(* CODESYS project festo_vtem_devcon_v3.5.7.235.library
   Version: 3.5.7.235
   Author: JEBU/MKLP
   Description: Festo VTEM device controlling functions interface
   Title: Festo_VTEM_DevCon
   DefaultNamespace: FestoVTEMdc
   LanguageModelAttribute: qualified-access-only
   Company: Festo SE & Co. KG

Project tree, tasks and I/O mapping:
  data type eValveState
  auxiliary Functions/
    function block FB_Read_Bits_From_Word [ST]
    function block FB_Write_Value_To_Word [ST]
    function block FB_Read_Bits_From_Byte [ST]
  StateInterpreter/
    function block FB_StateInterpreter_MA_07 [ST]
    function block FB_StateInterpreter_MA_01 [ST]
    function block FB_StateInterpreter_MA_11 [ST]
    function block FB_StateInterpreter_MA_12 [ST]
    function block FB_StateInterpreter_MA_06 [ST]
    function block FB_StateInterpreter_MA_02 [ST]
    function block FB_StateInterpreter_MA_03 [ST]
    function block FB_StateInterpreter_MA_04 [ST]
    function block FB_StateInterpreter_MA_05 [ST]
    function block FB_StateInterpreter_MA_08 [ST]
    function block FB_StateInterpreter_MA_33 [ST]
    function block FB_StateInterpreter_TeachInRun [ST]
  Operation/
    data type eResponseToValveModeSet
    function block FB_ValveControl [ST]
    function block FB_TeachInRun [ST]
  Transfermode/
    data type eTransferResponse
    data type stTransferPackage
    specific_MA_config/
      function block FB_Write_config_MA_07 [ST]
      function block FB_Write_config_MA_04 [ST]
      function block FB_Write_config_MA_11 [ST]
      function block FB_Write_config_MA_12 [ST]
      function block FB_Write_config_MA_02 [ST]
      function block FB_Write_config_MA_03 [ST]
      function block FB_Write_config_MA_08 [ST]
      function block FB_Write_config_MA_05 [ST]
      function block FB_Write_config_MA_01 [ST]
      function block FB_Write_config_MA_06 [ST]
      function block FB_Write_config_MA_33 [ST]
    data type eSavingResponse
    data type stMalfunction
    function block FB_Download_Multiple_Parameters [ST]
    function block FB_Download_Single_Parameter [ST]
    function block FB_Upload_Multiple_Parameters [ST]
    function block FB_Upload_Single_Parameter [ST]
    function block FB_Save_Configuration_Persistent [ST]
    function block FB_Write_config_AI_Module [ST]
    function block FB_Write_config_DI_Module [ST]
    function block FB_ReadMalfunctionList [ST]
  data type eValveMode
  data type eResponseTeachInRun
  data type eResponseReadMalfunctionList
*)

// Operation/eResponseToValveModeSet
(*****************************************************************************************************

Festo SE & Co. KG, Esslingen
Copyright (c) 2019. All rights reserved.

Product:            Motion Terminal VTEM
Description:        Enum for responding values sent by the Motion Terminal or the function blocks

Object version:     1.01
Last change:        2019
======================================================================================================
                                       H I S T O R Y
======================================================================================================
Version:            1.01
Date:               2019-04
Change/Activity:    - added new Value "FB_not_enabled := 1051"
Release:            3.5.7.232
Author:             MKLP
------------------------------------------------------------------------------------------------------
Version:            1.00
Date:               2017
Change/Activity:    - created
Release:            3.5.7.220
Author:             HLBG
======================================================================================================

*****************************************************************************************************)

TYPE eResponseToValveModeSet :
(
	// info provided by Motion Terminal protocol ("app state")
	reserved 								:= 0,
	invalid_SetValveMode 					:= 1,
	invalid_SetAppControl 					:= 2,
	invalid_SetAppOption 					:= 3,
	invalid_SetPointValue1 					:= 4,
	invalid_SetPointValue2 					:= 5,
	invalid_configuration 					:= 6,

	access_denied_WebConfig 				:= 10,
	access_denied_saving_parameterisation 	:= 11,
	no_license_for_this_MA 					:= 12,
	all_licenses_in_use 					:= 13,
	invalid_license_file 					:= 14,
	no_valve_detected 						:= 15,
	valve_self_calibration_running 			:= 16,
	

	// additional FB internal info (not part of Motion Terminal protocol)
	no_TransferMode_with_this_FB			:= 1020,
	
	preparing_for_start 					:= 1031,
	starting 								:= 1032,
	MA_running 								:= 1033,
	TransferMode_running					:= 1034,
	stopping 								:= 1035,
	all_MAs_stopped 						:= 1036,
	acknowledge_needed 						:= 1037,
	failure 								:= 1038,

	preparing_for_acknowledge 				:= 1040,
	acknowledging 							:= 1041,
	all_errors_acknowledged 				:= 1042,
	failure_still_active 					:= 1043,

	no_communication 						:= 1050,
	FB_not_enabled							:= 1051
);
END_TYPE

// eValveState
(*****************************************************************************************************

Festo SE & Co. KG, Esslingen
Copyright (c) 2018. All rights reserved.

Product:            Motion Terminal VTEM
Description:        Enum to interpret the valve state value

Object version:     1.00
Last change:        2017
======================================================================================================
                                       H I S T O R Y
======================================================================================================
Version:            1.00
Date:               2017
Change/Activity:    - created
Release:            3.5.7.220
Author:             HLBG
======================================================================================================

*****************************************************************************************************)

TYPE eValveState :
(
	// info provided by Motion Terminal protocol ("valve state")
	NotReady 		:= 0, 
	Configurable 	:= 1, 
	Running 		:= 2,
	Failure 		:= 3
);
END_TYPE

// Transfermode/eTransferResponse
(*****************************************************************************************************

Festo SE & Co. KG, Esslingen
Copyright (c) 2018. All rights reserved.

Product:            Motion Terminal VTEM
Description:        Enum for responding values sent by the Motion Terminal or the function blocks

Object version:     1.03
Last change:        2020-03
======================================================================================================
                                       H I S T O R Y
======================================================================================================
Version:            1.03
Date:               2020-03
Change/Activity:    - added value 8 (#3104444)
Release:            not released yet
Author:             JEBU/MKLP
------------------------------------------------------------------------------------------------------
Version:            1.02
Date:               2018-11
Change/Activity:    - added values 29, 30 
Release:            3.5.7.233
Author:             JEBU
------------------------------------------------------------------------------------------------------
Version:            1.01
Date:               2018-08
Change/Activity:    - added values 27, 28 
Release:            3.5.7.221
Author:             JEBU
------------------------------------------------------------------------------------------------------
Version:            1.00
Date:               2017
Change/Activity:    - created
Release:            3.5.7.220
Author:             HLBG
======================================================================================================

*****************************************************************************************************)

TYPE eTransferResponse :
(
	// info provided by Motion Terminal protocol ("invalid command")
	reserved 								:= 0,
	invalid_Channel 						:= 1,
	invalid_TransferControl 				:= 2,
	invalid_AddressedTarget 				:= 3,
	invalid_Index 							:= 4,
	invalid_TransferValue 					:= 5,
	invalid_Combination 					:= 6,
	access_denied_DataInUse					:= 7,
	no_data_empty_slot						:= 8,
	
	// additional FB internal info (not part of Motion Terminal protocol)
	invalid_ParameterSet 					:= 9,
	
	// info provided by Motion Terminal protocol ("app state")
	access_denied_WebConfig 				:= 10,
	access_denied_saving 					:= 11,
	no_valve_detected 						:= 15,
	
	// additional FB internal info (not part of Motion Terminal protocol)
	reading_transfermode					:= 20,	
	ready_for_new_transfer 					:= 21,
	preparing_transfer 						:= 22,
	transferring 							:= 23,
	transfer_successful 					:= 24,
	FB_needs_rising_edge_xExecute			:= 25,
	Valve_Mode_is_not_61_inactive			:= 26,
	invalid_firmware_version				:= 27,
	communication_failed					:= 28,
	invalid_module_number					:= 29,
	resetting								:= 30
);
END_TYPE

// Transfermode/stTransferPackage
(*****************************************************************************************************

Festo SE & Co. KG, Esslingen
Copyright (c) 2018. All rights reserved.

Product:            Motion Terminal VTEM
Description:        Struct for transfer mode data

Object version:     1.00
Last change:        2017
======================================================================================================
                                       H I S T O R Y
======================================================================================================
Version:            1.00
Date:               2017
Change/Activity:    - created
Release:            3.5.7.220
Author:             HLBG
======================================================================================================

*****************************************************************************************************)

TYPE stTransferPackage :
	STRUCT
		iChannel			: INT;		(* the channel the value is to be written to (see documentation for details) *)
		iAddressedTarget	: INT; 		(* the target by which the parameter value is to be used (was "iAddressedApp" in former versions) (see documentation for details)*)
		iIndex				: INT; 		(* the index of the parameter (see documentation for details) *)
		iTransferValue		: INT; 		(* the value to be transfered *)
	END_STRUCT
END_TYPE

// Transfermode/eSavingResponse
(*****************************************************************************************************

Festo SE & Co. KG, Esslingen
Copyright (c) 2018. All rights reserved.

Product:            Motion Terminal VTEM
Description:        Enum for values sent back from the Motion Terminal during saving process 

Object version:     1.01
Last change:        2019-07
======================================================================================================
                                       H I S T O R Y
======================================================================================================
Version:            1.01
Date:               2019-07
Change/Activity:    - added value 25 "FB_needs_rising_edge_xExecute" (#2369163)
Release:            not released yet
Author:             JEBU/MKLP
------------------------------------------------------------------------------------------------------
Version:            1.00
Date:               2017
Change/Activity:    - created
Release:            3.5.7.220
Author:             HLBG
======================================================================================================

*****************************************************************************************************)

TYPE eSavingResponse :
(
	// info provided by Motion Terminal protocol (saving progress)
	reserved 				:= 0,
	saving_in_progress 		:= 1,
	saving_successful 		:= 2,
	saving_not_possible 	:= 3,
	saving_failed 			:= 4,
	
	// info provided by Motion Terminal protocol ("app state")
	access_denied_WebConfig := 10,
	access_denied_saving	:= 11,
	no_valve_detected 		:= 15,
	
	// additional FB internal info (not part of Motion Terminal protocol)
	preparing_to_save 		:= 20,
	ready_to_save 			:= 21,
	FB_needs_rising_edge_xExecute	:= 25
);
END_TYPE

// eValveMode
(*****************************************************************************************************

Festo SE & Co. KG, Esslingen
Copyright (c) 2018. All rights reserved.

Product:            Motion Terminal VTEM
Description:        Enum for values of the valve mode 

Object version:     1.01
Last change:        2020-04
======================================================================================================
                                       H I S T O R Y
======================================================================================================
Version:            1.01
Date:               2020-04
Change/Activity:    - created
Release:            3.5.7.234
Author:             JEBU
======================================================================================================

*****************************************************************************************************)

TYPE eValveMode :
(
	MA01_Directional_control_valve_functions							:= 1,
	MA02_Proportional_directional_control_valve							:= 2,
	MA03_Proportional_pressure_regulation								:= 3,
	MA04_Modelbased_proportional_pressure_regulation					:= 4,
	MA05_Supply_and_exhaust_air_flow_control							:= 5,
	MA06_ECO_drive														:= 6,
	MA07_Presetting_of_travel_time										:= 7,
	MA08_Selectable_pressure_level_ECO									:= 8,
	MA11_Soft_stop														:= 11,
	MA12_Leakage_diagnostics											:= 12,
	MA32_Positioning_and_Force											:= 32,
	MA33_Positioning													:= 33,
	VM60_TeachIn_run													:= 60,
	VM61_Inactive														:= 61,
	VM63_Transfermode													:= 63
);
END_TYPE

// Transfermode/stMalfunction
(*****************************************************************************************************

Festo SE & Co. KG, Esslingen
Copyright (c) 2018. All rights reserved.

Product:            Motion Terminal VTEM
Description:        Struct for complete entry in malfunction list (code, subcode, classification)

Object version:     1.00
Last change:        2018
======================================================================================================
                                       H I S T O R Y
======================================================================================================
Version:            1.00
Date:               2018
Change/Activity:    - created (#2256305)
Release:            not released yet
Author:             JEBU
======================================================================================================

*****************************************************************************************************)

TYPE stMalfunction :
STRUCT
	usiMalfunctionCode				: USINT;		// Malfunction Code
	usiMalfunctionSubcode			: USINT;		// Malfunction Subcode
	usiMalfunctionClassification	: USINT;		// Malfunction Classification
END_STRUCT
END_TYPE

// eResponseTeachInRun
(*****************************************************************************************************

Festo SE & Co. KG, Esslingen
Copyright (c) 2019. All rights reserved.
 
Product:            Motion Terminal VTEM
Description:        Enum status of the teach-in run process as it is displayed in the app state byte
 
Object version:     1.05
Last change:        2020-04
======================================================================================================
                                       H I S T O R Y
======================================================================================================
Version:            1.05
Date:               2020-04
Change/Activity:    - created (#2256363)
Release:            3.5.7.234
Author:             JEBU
======================================================================================================

******************************************************************************************************)

TYPE eResponseTeachInRun :
(
	// following entries correspond to the values of the AppState byte of the teach-in run
	TeachInRun_reserved								:= 0,
	TeachInRun_unlearned							:= 1,
	TeachInRun_check_tubes							:= 2,
	TeachInRun_choose_control						:= 3,
	TeachInRun_tune_trajectory						:= 4,
	TeachInRun_determine_reference_value			:= 5,
	TeachInRun_identification						:= 6,
	TeachInRun_partially_completed_only_2			:= 12,
	TeachInRun_partially_completed_only_4			:= 13,
	TeachInRun_completed							:= 14,
	TeachInRun_error								:= 15,
	
	// following entries are copies from eResponseToValveModeSet, their values are origins + 100	
	invalid_SetValveMode 							:= 101,
	invalid_SetAppControl 							:= 102,
	invalid_SetAppOption 							:= 103,
	invalid_SetPointValue1 							:= 104,
	invalid_SetPointValue2 							:= 105,
	invalid_configuration 							:= 106,
                                            	
	access_denied_WebConfig 						:= 110,
	access_denied_saving_parameterisation 			:= 111,
	no_license_for_this_MA 							:= 112,
	all_licenses_in_use 							:= 113,
	invalid_license_file 							:= 114,
	no_valve_detected 								:= 115,
	valve_self_calibration_running 					:= 116,
	
	// additional FB internal info (not part of Motion Terminal protocol)
	idle											:= 210,
	storing_first_cycle_input_data					:= 215,
	resetting_valve_to_61							:= 220,
	ReadingActiveParameterSet						:= 230,
	ChangingActiveParameterSet						:= 232,
	writing_parameter_MotionAppToBeToughtIn			:= 234,
	running_teachIn_run								:= 240,
	error_occured_check_DiagnosticMemory			:= 270,
	input_data_invalid								:= 271,
	FB_needs_rising_edge_xEnable					:= 272,
	acknowledge_needed								:= 273,
	Invalid_MotionAppToBeToughtIn					:= 274,
	resetting										:= 300	
);
END_TYPE

// eResponseReadMalfunctionList
(*****************************************************************************************************

Festo SE & Co. KG, Esslingen
Copyright (c) 2018. All rights reserved.

Product:            Motion Terminal VTEM
Description:        This enum contains the values for the response output of the FB_ReadMalfunctionList

Object version:     1.00
Last change:        2020-03
======================================================================================================
                                       H I S T O R Y
======================================================================================================
Version:            1.00
Date:               2019
Change/Activity:    - created (#2256305)
Release:            3.5.7.234
Author:             JEBU/MKLP
======================================================================================================

*****************************************************************************************************)


TYPE eResponseReadMalfunctionList :
(
	// function block specific repsonse
		idle									:= 0,
		setting_valve_to_inactive				:= 1,
		getting_malfunction_count				:= 2,
		transferring 							:= 3,
		done									:= 4,
		no_entries_in_malfunction_list			:= 5,
		error_while_transmitting_data_to_vtem	:= 6,
		aborting								:= 7,
		resetting								:= 8,
		
		FB_needs_rising_edge_xExecute			:= 10,
	//-------------------------------------------------------------------------------------

	// info provided by Motion Terminal protocol ("app state") with an offset of +100
		reserved 								:= 100,
		invalid_SetValveMode 					:= 101,
		invalid_SetAppControl 					:= 102,
		invalid_SetAppOption 					:= 103,
		invalid_SetPointValue1 					:= 104,
		invalid_SetPointValue2 					:= 105,
		invalid_configuration 					:= 106,
		
		access_denied_WebConfig 				:= 110,
		access_denied_saving_parameterisation 	:= 111,
		no_license_for_this_MA 					:= 112,
		all_licenses_in_use 					:= 113,
		invalid_license_file 					:= 114,
		no_valve_detected 						:= 115,
		valve_self_calibration_running 			:= 116,
	//-------------------------------------------------------------------------------------

	// info provided by Motion Terminal protocol ("invalid command transfer mode") with an offset of +200
		invalid_Channel 						:= 201,
		invalid_TransferControl 				:= 202,
		invalid_iChooseOtherValve				:= 203,	// invalid_AddressedTarget is always invalid_iChooseOtherValve
		invalid_Index 							:= 204,
		invalid_TransferValue 					:= 205,
		no_valve_detected_at_selected_slot 		:= 206,	// invalid_Combination is always no_valve_detected_at_selected_slot
		access_denied_DataInUse					:= 207,
		no_data_empty_slot						:= 208
	//-------------------------------------------------------------------------------------
);
END_TYPE

// StateInterpreter/FB_StateInterpreter_MA_07
/// The variable "byActualAppState" is an output of the FB_ValveControl that is used differently in each Motion App.
/// This function block interprets the "AppState" output of the FB_ValveControl if Motion App 7 ("Presetting of travel time") is running.
/// The Motion App specific values are derived from the "byActualAppState".

FUNCTION_BLOCK FB_StateInterpreter_MA_07
VAR_INPUT
	byActualAppState 		: BYTE; 	(* output of the FB_ValveControl *)
END_VAR                 	
VAR_OUTPUT              	
	xRetractedEndPos		: BOOL;  	(* indicates whether the retracted end position was reached (after outlet port 2 is pressurised) *)
	xAdvancedEndPos			: BOOL;  	(* indicates whether the advanced end position was reached (after outlet port 4 is pressurised) *)
	xWarning				: BOOL; 	(* indicates whether there is a warning returned by the Motion App *)
END_VAR                 	
VAR                     	
	fbReadBitsFromByte		: FB_Read_Bits_From_Byte; 
	byRetractedEndPos		: BYTE;
	byAdvancedEndPos		: BYTE;
	byWarning				: BYTE;
END_VAR

(*****************************************************************************************************

Festo SE & Co. KG, Esslingen
Copyright (c) 2018. All rights reserved.

Product:            Motion Terminal VTEM
Description:        Function block for interpreting the app state of Motion App 7 

Object version:     1.00
Last change:        2017
======================================================================================================
                                       H I S T O R Y
======================================================================================================
Version:            1.00
Date:               2017
Change/Activity:    - created
Release:            3.5.7.220
Author:             HLBG
======================================================================================================

*****************************************************************************************************)

// read the Motion App specific values from the ActualAppState byte
fbReadBitsFromByte(byData := byActualAppState, iStartBit := 0, iEndBit := 0, byValue => byRetractedEndPos);
xRetractedEndPos :=  BYTE_TO_BIT(byRetractedEndPos);

fbReadBitsFromByte(byData := byActualAppState, iStartBit := 2, iEndBit := 2, byValue => byAdvancedEndPos); 
xAdvancedEndPos :=  BYTE_TO_BIT(byAdvancedEndPos);

fbReadBitsFromByte(byData := byActualAppState, iStartBit := 7, iEndBit := 7, byValue => byWarning);
xWarning := BYTE_TO_BIT(byWarning);

END_FUNCTION_BLOCK

// Operation/FB_ValveControl
/// This is the central function block for the operation of Motion Apps on a valve. 
/// The FB serves to operate all Motion Apps with their specific setpoint values.  
/// It is able to execute and to stop Motion Apps and to deal with occuring errors. 
/// Parameterisation is not possible with this function block.

FUNCTION_BLOCK FB_ValveControl
VAR_INPUT
	awBusDataFromVTEM			: ARRAY[0..2] OF WORD;		(* 6 bytes of process data that is received from the Motion Terminal *)
END_VAR

VAR_IN_OUT
	awBusDataToVTEM				: ARRAY [0..2] OF WORD;		(* 6 bytes of process data that is sent to the Motion Terminal *)
END_VAR

VAR_INPUT
	xEnable						: BOOL; 					(* has to be set to TRUE in order to operate a Motion App on the valve, otherwise any motion is stopped *)	

	bySetValveMode				: BYTE; 					(* ID of the Motion App to be executed, 60 for 'commissioning', '61 for 'stop', 62 for 'acknowledge' *)
	bySetAppControl 			: BYTE; 					(* SetAppControl of the chosen bySetMode, see documentation of the valve mode for its meaning *)
	bySetAppOption 				: BYTE;						(* SetAppOption of the chosen bySetMode, see documentation of the valve mode for its meaning *)
	iSetpointValue1 			: INT; 						(* SetPoint1 of the chosen bySetMode, see documentation of the valve mode for its meaning *)
	iSetpointValue2 			: INT; 						(* SetPoint2 of the chosen bySetMode, see documentation of the valve mode for its meaning *)

	xManualAcknowledge			: BOOL;  					(* errors can be acknowledged (after they got inactive) with a rising edge at this input *)
END_VAR                     	

VAR_OUTPUT                  	
	byActualValveMode 			: BYTE; 					(* actual valve mode of the Motion Terminal *)
	byActualValveState 			: BYTE; 					(* actual valve state of the Motion Terminal *)
	byActualAppState 			: BYTE; 					(* Byte1 of the received process data: app state of the desired Motion App, see documentation of the valve mode for its meaning *)
	iActualValue1 				: INT;	 					(* ActualValue1 of the desired Motion App, see documentation of the valve mode for its meaning *)
	iActualValue2 				: INT;						(* ActualValue2 of the desired Motion App, see documentation of the valve mode for its meaning *)
	iResponseToValveModeSet		: eResponseToValveModeSet; 	(* enumeration that indicates the status of execution of the desired valve mode *)
	iErrorCode					: INT := 0; 				(* contains the malfunction code of the latest error, 0 if no error occurred so far *)
END_VAR                     	
VAR                         	
	aw_OperationCommand			: ARRAY [0..2] OF WORD;
	fbWriteValueToWord 			: FB_Write_Value_To_Word;
	fbReadBitsFromWord 			: FB_Read_Bits_From_Word;
	iCommandNumber				: INT;						(* control variable for the state machine *)
	iInvalidCommand				: INT;
	iRecChannel					: INT;
	iRecTransferCtrl			: INT;
	iRecAddressedTargetType		: INT;
	iRecIndex					: INT;
	iRecTransferValue			: INT;
	iActualValveMode			: INT;
	iValveState					: INT;

	xInvalidInput				: BOOL;
	xLastManualAcknowledge		: BOOL;
	xAcknowledging_in_progress 	: BOOL;						(* internal variable that indicates that an acknowledge process has been started *)
	
	xMalfunctionReading_Done	: BOOL := FALSE;
	iMalfunctionListEntry		: INT;
	iRecMalfunctionCode			: INT;
	iRecMalfunctionRating		: INT;
	iActualAppState				: INT;
END_VAR

(*****************************************************************************************************

Festo SE & Co. KG, Esslingen
Copyright (c) 2019. All rights reserved.

Product:            Motion Terminal VTEM
Description:        Function block to operate Motion Apps on the Motion Terminal VTEM

Object version:     2.02
Last change:        2019-11
======================================================================================================
                                       H I S T O R Y
======================================================================================================
Version:            2.02
Date:               2019-11
Change/Activity:    - FB detect a falling edge of xManualAcknowledge while input xEnable is FALSE
Release:            3.5.7.234
Author:             MKLP
------------------------------------------------------------------------------------------------------
Version:            2.01
Date:               2019-04
Change/Activity:    - setting iResponseToValveModeSet to "FB_not_enabled" when then FB is not enabled
					(#2417678)
                    - updated enable = FALSE behaviour
Release:            3.5.7.232
Author:             MKLP
------------------------------------------------------------------------------------------------------
Version:            2.00
Date:               2019-03
Change/Activity:    - changed output awBusDataToVTEM to VAR_IN_OUT (#2368965)
Release:            3.5.7.230
Author:             JEBU
------------------------------------------------------------------------------------------------------
Version:            1.02
Date:               2018-11
Change/Activity:    - fixed bug related to invalid app control (#2173876)
Release:            3.5.7.221
Author:             JEBU
------------------------------------------------------------------------------------------------------
Version:            1.01
Date:               2018-08
Change/Activity:    - changed behavior of invalid app control
Release:            3.5.7.220
Author:             JEBU
------------------------------------------------------------------------------------------------------
Version:            1.00
Date:               2017
Change/Activity:    - created
Release:            not released
Author:             HLBG
======================================================================================================

*****************************************************************************************************)

// read the protocol data of the Motion Terminal
	fbReadBitsFromWord(wData := awBusDataFromVTEM[0], iStartBit := 0, iEndBit := 5, iValue => iActualValveMode);
	byActualValveMode := INT_TO_BYTE(iActualValveMode);
	fbReadBitsFromWord(wData := awBusDataFromVTEM[0], iStartBit := 6, iEndBit := 7, iValue => iValveState);
	byActualValveState := INT_TO_BYTE(iValveState);
	fbReadBitsFromWord(wData := awBusDataFromVTEM[0], iStartBit := 8, iEndBit := 15, iValue => iActualAppState);
	byActualAppState := INT_TO_BYTE(iActualAppState);
	
	iActualValue1 := WORD_TO_INT(awBusDataFromVTEM[1]);
	iActualValue2 := WORD_TO_INT(awBusDataFromVTEM[2]);

IF xEnable = FALSE AND ((iActualValveMode = 61 AND iResponseToValveModeSet <> eResponseToValveModeSet.stopping) OR iActualValveMode = 63 OR iCommandNumber = 0) THEN	// goto idle state
	IF iActualValveMode = 63 AND iResponseToValveModeSet <> eResponseToValveModeSet.FB_not_enabled THEN 	// Exit the TM if it is running while the falling edge of xEnable
		iCommandNumber := 4;	// exit TransferMode
	ELSIF iActualValveMode = 61 AND iCommandNumber <>2 AND iCommandNumber <> 0 AND iResponseToValveModeSet <> eResponseToValveModeSet.FB_not_enabled THEN	//Ensure that the last command is iCommandNumber = 2 (Stop)
		iCommandNumber := 2;	// do nothing (here: command 'stop' to ensure the valve remains stopped and it is the last command the FB sends)
	ELSE // IDLE-State: repeated during xEnable = FALSE
		iCommandNumber := 0;	// IDLE - FB stops overwritting Busdata
		iResponseToValveModeSet := eResponseToValveModeSet.FB_not_enabled;
	END_IF

ELSE
	// pre-check of the state of the Motion Terminal
	IF byActualValveMode = 0 AND byActualValveState = eValveState.NotReady THEN							 	// The communication to the Motion Terminal has been lost
		iResponseToValveModeSet :=  eResponseToValveModeSet.no_communication;
		iCommandNumber := 2; 	// do nothing (here: command 'stop' to ensure the valve remains stopped)
	ELSIF byActualValveMode = 61 AND byActualAppState = 10 THEN 											// The WebConfig has write permission -> access denied for the PLC
		iResponseToValveModeSet :=  eResponseToValveModeSet.access_denied_WebConfig;
		iCommandNumber := 2; 	// do nothing (here: command 'stop' to ensure the valve remains stopped)
	ELSIF byActualValveMode = 61 AND byActualAppState = 11 THEN 											// A saving process is executed -> access denied for the PLC
		iResponseToValveModeSet :=  eResponseToValveModeSet.access_denied_saving_parameterisation;
		iCommandNumber := 2; 	// do nothing (here: command 'stop' to ensure the valve remains stopped)
	ELSIF byActualValveMode = 61 AND byActualAppState = 15 THEN												// no valve was detected at the addressed slot
		iResponseToValveModeSet :=  eResponseToValveModeSet.no_valve_detected;
		iCommandNumber := 2; 	// do nothing (here: command 'stop' to ensure the valve remains stopped)
	
	// end of pre-check, verification of the desired command
	ELSIF xEnable = TRUE AND bySetValveMode > 0 AND bySetValveMode < 61 THEN								// A Motion App is to be executed
		// checking the data range for the input value BySetAppControl
		IF bySetAppControl < 0 OR bySetAppControl > 3 THEN
			xInvalidInput := TRUE;
			iResponseToValveModeSet := eResponseToValveModeSet.invalid_SetAppControl;
		ELSE
			xInvalidInput := FALSE;
		END_IF;
	
		// analysis of the state of the Motion Terminal and definition of the specific reaction (= command to the Motion Terminal)
		IF xInvalidInput = TRUE THEN
			iCommandNumber := 2;		// command 'stop'
			
		ELSIF byActualValveState = eValveState.RUNNING AND byActualValveMode = bySetValveMode THEN				// The desired Motion App is already running
			iCommandNumber := 1;		// operation of the Motion App
			iResponseToValveModeSet := eResponseToValveModeSet.MA_running;
	
		ELSIF byActualValveState = eValveState.RUNNING AND byActualValveMode <> bySetValveMode THEN			// A Motion App is running but it is not the desired one
			iCommandNumber := 2;  		// command 'stop' (stopping the other MA in order to start the desired MA)
			iResponseToValveModeSet := eResponseToValveModeSet.preparing_for_start;
					
		ELSIF byActualValveState = eValveState.Configurable AND byActualValveMode = 61 THEN					// The valve is ready to operate a Motion App
			// ( A Motion App was stopped or an error was acknowledged to reach this state )
			iCommandNumber := 1; 				// operate the Motion App
			xAcknowledging_in_progress := FALSE;
		
			// check whether the Motion App didn't start due to an invalid command
			fbReadBitsFromWord(wData := awBusDataFromVTEM[0], iStartBit := 8, iEndBit := 15, iValue => iInvalidCommand);
			// creating the ResponseToValveModeSet in dependency of the "InvalidCommand" value
			IF iInvalidCommand = 0 THEN
				iResponseToValveModeSet := eResponseToValveModeSet.starting; 			// no invalid command
			ELSIF iInvalidCommand = 1 THEN
				iResponseToValveModeSet := eResponseToValveModeSet.invalid_SetValveMode;
			ELSIF iInvalidCommand = 2 THEN
				iResponseToValveModeSet := eResponseToValveModeSet.invalid_SetAppControl;
			ELSIF iInvalidCommand = 3 THEN
				iResponseToValveModeSet := eResponseToValveModeSet.invalid_SetAppOption;
			ELSIF iInvalidCommand = 4 THEN
				iResponseToValveModeSet := eResponseToValveModeSet.invalid_SetPointValue1;
			ELSIF iInvalidCommand = 5 THEN
				iResponseToValveModeSet := eResponseToValveModeSet.invalid_SetPointValue2;
			ELSIF iInvalidCommand = 6 THEN
				iResponseToValveModeSet := eResponseToValveModeSet.invalid_configuration;
			ELSIF iInvalidCommand = 10 THEN
	 			iResponseToValveModeSet := eResponseToValveModeSet.access_denied_WebConfig;
			ELSIF iInvalidCommand = 11 THEN
	 			iResponseToValveModeSet := eResponseToValveModeSet.access_denied_saving_parameterisation;
			ELSIF iInvalidCommand = 12 THEN
				iResponseToValveModeSet := eResponseToValveModeSet.no_license_for_this_MA;
			ELSIF iInvalidCommand = 13 THEN
				iResponseToValveModeSet := eResponseToValveModeSet.all_licenses_in_use;
			ELSIF iInvalidCommand = 14 THEN
				iResponseToValveModeSet := eResponseToValveModeSet.invalid_license_file;
			ELSIF iInvalidCommand = 15 THEN
				iResponseToValveModeSet := eResponseToValveModeSet.no_valve_detected;
			ELSIF iInvalidCommand = 16 THEN
				iResponseToValveModeSet := eResponseToValveModeSet.valve_self_calibration_running;
			END_IF
					
		ELSIF byActualValveState = eValveState.Configurable AND byActualValveMode = 63 THEN					// The valve is using the transfer mode for parameterisation
			iCommandNumber := 4; 	// command 'exit transfer mode'
			iResponseToValveModeSet := eResponseToValveModeSet.preparing_for_start;
			xAcknowledging_in_progress := FALSE;
					
		ELSIF (byActualValveState = eValveState.Failure OR byActualValveState = eValveState.NotReady)  AND (byActualValveMode <> 63) THEN 		// An error occurred -> read the malfunction code
			IF xMalfunctionReading_Done = FALSE THEN
				iMalfunctionListEntry := 1;
				iCommandNumber := 3; 		// command 'read malfunction code'
			ELSE	// The error has already been read -> no further action, wait for acknowledge
				iCommandNumber := 2; 		// command 'stop'
			END_IF
			
			// create the ResponseToValveModeSet
			IF byActualValveState = eValveState.Failure THEN
				iResponseToValveModeSet := eResponseToValveModeSet.Failure;
				xAcknowledging_in_progress := FALSE;
			ELSE	//byActualValveState = Not Ready
				iResponseToValveModeSet := eResponseToValveModeSet.acknowledge_needed;
			END_IF
				
		ELSIF (byActualValveState = eValveState.Failure OR byActualValveState = eValveState.NotReady) AND byActualValveMode = 63 THEN			// An error occurred and the Motion Terminal already switched to transfer mode in order to read the malfunction code
			// create the ResponseToValveModeSet
			IF byActualValveState = eValveState.Failure THEN
				iResponseToValveModeSet := eResponseToValveModeSet.failure;
				xAcknowledging_in_progress := FALSE;
			ELSE
				iResponseToValveModeSet := eResponseToValveModeSet.acknowledge_needed;
			END_IF
			
		
			// read the transfer mode variables from status data
			fbReadBitsFromWord(wData := awBusDataFromVTEM[0], iStartBit := 8, iEndBit := 12, iValue => iRecChannel);
			fbReadBitsFromWord(wData := awBusDataFromVTEM[0], iStartBit := 13, iEndBit := 15, iValue => iRecTransferCtrl);
			fbReadBitsFromWord(wData := awBusDataFromVTEM[1], iStartBit := 0, iEndBit := 5, iValue => iRecAddressedTargetType);
			fbReadBitsFromWord(wData := awBusDataFromVTEM[1], iStartBit := 8, iEndBit := 15, iValue => iRecIndex);
			
						
			IF iRecChannel = 31 AND iRecTransferCtrl = 2 AND iRecAddressedTargetType = 0 AND iRecIndex = iMalfunctionListEntry THEN
				// The specified entry of the malfunction list was read
				fbReadBitsFromWord(wData := awBusDataFromVTEM[2], iStartBit := 0, iEndBit := 7, iValue => iRecMalfunctionCode);
	 			fbReadBitsFromWord(wData := awBusDataFromVTEM[2], iStartBit := 14, iEndBit := 15, iValue => iRecMalfunctionRating);
				
				IF iRecMalfunctionRating = 1 (* active error *) OR iRecMalfunctionRating = 2 (* inactive error *) THEN
					// The error was read correctly
					iCommandNumber := 4; 	// command 'exit transfer mode'
					iErrorCode := iRecMalfunctionCode;
					xMalfunctionReading_Done := TRUE;
					
				ELSIF iRecMalfunctionRating = 3 (* warning *) THEN
					// The entry is a warning -> read next entry to find an error
					iMalfunctionListEntry := iMalfunctionListEntry +1;
					iCommandNumber := 3; 	// command 'read malfunction code'
					
				ELSE	// iRecMalfunctionRating = 0 -> no valid entry in malfunction list
					// no entry available in the malfunction list
					iCommandNumber := 4; 	// command 'exit transfer mode'
	 				xMalfunctionReading_Done := TRUE;
				END_IF; 
	 				
			ELSE	// NOT the specified entry of the malfunction list was read
				IF xMalfunctionReading_Done = FALSE THEN
					iMalfunctionListEntry := 1; 
					iCommandNumber := 3; 		// command 'read malfunction code' 
				ELSE
					iCommandNumber := 4; 		// command 'exit transfer mode'
				END_IF
			END_IF
		END_IF
						
	ELSIF (xEnable = FALSE AND bySetValveMode > 0 AND bySetValveMode < 61) OR bySetValveMode = 61 THEN		// stop all Motion Apps
		IF byActualValveState = eValveState.Configurable OR byActualValveState = eValveState.Running THEN
			xAcknowledging_in_progress := FALSE;
			IF byActualValveMode = 61 THEN			// all Motion Apps stopped
				iResponseToValveModeSet := eResponseToValveModeSet.all_MAs_stopped;
				iCommandNumber := 2; 	// command 'stop'
			ELSIF byActualValveMode = 63 THEN		// transfer mode is active
				iResponseToValveModeSet := eResponseToValveModeSet.all_MAs_stopped;
				iCommandNumber := 4; 	// command 'exit transfer mode'
			ELSE	// Motion App is active
				iResponseToValveModeSet := eResponseToValveModeSet.stopping;
				iCommandNumber := 2; 	// command 'stop'
			END_IF
				
		ELSE // (byActualValveState = eValveState.NotReady OR byActualValveState = eValveState.Failure)
			// keep the valve stopped and read the error
			IF byActualValveState = eValveState.Failure THEN
				iResponseToValveModeSet := eResponseToValveModeSet.failure; 
				xAcknowledging_in_progress := FALSE; 
			ELSE
				iResponseToValveModeSet := eResponseToValveModeSet.acknowledge_needed; 
			END_IF
			
			IF byActualValveMode <> 63 THEN
				// define the command to be sent to the Motion Terminal
				IF xMalfunctionReading_Done = FALSE THEN
					iMalfunctionListEntry := 1;
					iCommandNumber := 3; 		// command 'read malfunction code'
				ELSE
					iCommandNumber := 2; 		// command 'stop'
				END_IF
			ELSE // byActualValveMode = 63
				// read the transfer variables from the status data
				fbReadBitsFromWord(wData := awBusDataFromVTEM[0], iStartBit := 8, iEndBit := 12, iValue => iRecChannel);
				fbReadBitsFromWord(wData := awBusDataFromVTEM[0], iStartBit := 13, iEndBit := 15, iValue => iRecTransferCtrl);
				fbReadBitsFromWord(wData := awBusDataFromVTEM[1], iStartBit := 0, iEndBit := 5, iValue => iRecAddressedTargetType);
				fbReadBitsFromWord(wData := awBusDataFromVTEM[1], iStartBit := 8, iEndBit := 15, iValue => iRecIndex);
							
				IF iRecChannel = 31 AND iRecTransferCtrl = 2 AND iRecAddressedTargetType = 0 AND iRecIndex = iMalfunctionListEntry THEN
					// The specified entry of the malfunction list was read
					fbReadBitsFromWord(wData := awBusDataFromVTEM[2], iStartBit := 0, iEndBit := 7, iValue => iRecMalfunctionCode);
					fbReadBitsFromWord(wData := awBusDataFromVTEM[2], iStartBit := 14, iEndBit := 15, iValue => iRecMalfunctionRating);
					
					IF iRecMalfunctionRating = 1 (* active error *) OR iRecMalfunctionRating = 2 (* inactive error *) THEN
						iCommandNumber := 4; 	// command 'exit transfer mode'
						iErrorCode := iRecMalfunctionCode;
						xMalfunctionReading_Done := TRUE;
						
					ELSIF iRecMalfunctionRating = 3 (* warning *) THEN
						// The entry is a warning, reading next entry to find an error
						iMalfunctionListEntry := iMalfunctionListEntry +1;
						iCommandNumber := 3; 	// command 'read malfunction code'
					ELSE	// iRecMalfunctionRating = 0 -> no valid entry in malfunction list
						iCommandNumber := 4; 	// command 'exit transfer mode'
						xMalfunctionReading_Done := TRUE;
					END_IF
				
				ELSE	// NOT the specified entry of the malfunction list was read
					IF xMalfunctionReading_Done = FALSE THEN
						iMalfunctionListEntry := 1;
						iCommandNumber := 3; 		// command 'read malfunction code'
					ELSE
						iCommandNumber := 4; 		// command 'exit transfer mode'
					END_IF
				END_IF
			END_IF
	
		END_IF
		
	ELSIF bySetValveMode = 62 THEN																			// acknowledge (inactive) errors
		xMalfunctionReading_Done := FALSE;		// with this valve mode the malfunction list is reset
		iErrorCode := 0;
		IF byActualValveState = eValveState.Running THEN
			// A Motion App is running, no errors that have to be acknowledged
			iResponseToValveModeSet := eResponseToValveModeSet.all_errors_acknowledged;
			iCommandNumber := 2; 	// command 'stop' as no app activity is allowed in acknowledge mode
				
		ELSIF byActualValveState = eValveState.Configurable THEN
			// valve is ready, no errors that have to be acknowledged
			iResponseToValveModeSet :=  eResponseToValveModeSet.all_errors_acknowledged;
			iCommandNumber := 2; 	// do nothing (here: command 'stop' to remain in this state)
				
		ELSIF byActualValveState = eValveState.notReady THEN
			// The error is not active any more
			IF byActualValveMode = 63 THEN
				// valve is in transfer mode
				iResponseToValveModeSet := eResponseToValveModeSet.preparing_for_acknowledge ; 
				iCommandNumber := 4;	// command 'exit transfer mode'
			ELSE
				// The error can be acknowledged
				iResponseToValveModeSet :=  eResponseToValveModeSet.acknowledging;
				iCommandNumber := 5; 	// command 'acknowledge'
			END_IF
				
		ELSIF byActualValveState = eValveState.Failure THEN
			// The error is still active, therefore it cannot be acknowledged
			iResponseToValveModeSet := eResponseToValveModeSet.failure_still_active;
			iCommandNumber := 2; 	// do nothing (here: command 'stop', as the Motion App is already stopped due to failure) 
		END_IF
		
	
	ELSIF bySetValveMode = 63 THEN																			// 63 (transfer mode) not possible with this FB
		// no use of transfer mode in this function block possible due to missing input values (channel, index, etc.)
		iResponseToValveModeSet := eResponseToValveModeSet.no_TransferMode_with_this_FB;
		iCommandNumber := 2; 	// command 'stop'
		IF byActualValveState = eValveState.Configurable OR byActualValveState = eValveState.Failure THEN
			xAcknowledging_in_progress := FALSE;
		END_IF
		
	ELSE	// no valid valve mode
		iResponseToValveModeSet := eResponseToValveModeSet.invalid_SetValveMode;
		iCommandNumber := 2; 	// command 'stop'
		IF byActualValveState = eValveState.Configurable OR byActualValveState = eValveState.Failure THEN
			xAcknowledging_in_progress := FALSE;
		END_IF
	END_IF

	// If the Motion Terminal's state indicates acknowledgable errors (ValveState = NotReady), 
	// the input xManualAcknowledge is analysed to verify if the error can be acknowledged.
	// In this case the commands stated above are overwritten by the 'acknowledge' command.
	
	IF byActualValveState = eValveState.NotReady AND ((xManualAcknowledge = TRUE AND xLastManualAcknowledge = FALSE) OR (xAcknowledging_in_progress = TRUE)) THEN
		// There are errors that can be acknowledged AND the input values demand to acknowledge the error.
		// (rising edge at xManualAcknowledge)
		
		xMalfunctionReading_Done := FALSE;		// the malfunction list is reset
		iErrorCode := 0;
		
		IF byActualValveMode = 0 THEN			// no communication -> do nothing
			;
		ELSIF byActualValveMode = 63 THEN		// transfer mode is active
			xAcknowledging_in_progress := TRUE;
			iCommandNumber := 4; 		// command 'exit transfer mode'
			iResponseToValveModeSet := eResponseToValveModeSet.preparing_for_acknowledge;
		ELSE
			xAcknowledging_in_progress := TRUE;
			iCommandNumber := 5; 		// command 'acknowledge'
			iResponseToValveModeSet := eResponseToValveModeSet.acknowledging;
		END_IF
	END_IF
END_IF
xLastManualAcknowledge := xManualAcknowledge;

CASE iCommandNumber OF
	0:	// idle
	
	1:	// operation of the Motion App
		// create the operation command
		fbWriteValueToWord(iValue := bySetValveMode, iStartBit := 0, iEndBit := 5, wDataWord := awBusDataToVTEM[0]); 			// bySetValveMode
		fbWriteValueToWord(iValue := bySetAppControl, iStartBit := 6, iEndBit := 7, wDataWord := awBusDataToVTEM[0]); 			// bySetAppControl 
		fbWriteValueToWord(iValue := bySetAppOption, iStartBit := 8, iEndBit := 15, wDataWord := awBusDataToVTEM[0]); 			// bySetAppOption
		
		awBusDataToVTEM[1] := INT_TO_WORD(iSetpointValue1);
		awBusDataToVTEM[2] := INT_TO_WORD(iSetpointValue2);
		
	2: 	// command 'stop'
		fbWriteValueToWord(iValue := 61, iStartBit := 0, iEndBit := 5, wDataWord := awBusDataToVTEM[0]); 						// ValveMode = 61
		fbWriteValueToWord(iValue := 0, iStartBit := 6, iEndBit := 15, wDataWord := awBusDataToVTEM[0]); 						// (empty)

		awBusDataToVTEM[1] := 0; 																								// (empty)
		awBusDataToVTEM[2] := 0; 																								// (empty)

	3: 	// read the first malfunction code in transfer mode
		fbWriteValueToWord(iValue := 63, iStartBit := 0, iEndBit := 5, wDataWord := awBusDataToVTEM[0]); 						// ValveMode = 63
		fbWriteValueToWord(iValue := 0, iStartBit := 6, iEndBit := 7, wDataWord := awBusDataToVTEM[0]); 						// (empty)
		fbWriteValueToWord(iValue := 31, iStartBit := 8, iEndBit := 12, wDataWord := awBusDataToVTEM[0]); 						// Channel = 31
		fbWriteValueToWord(iValue := 2, iStartBit := 13, iEndBit := 15, wDataWord := awBusDataToVTEM[0]); 						// TransferCtrl = 2 (upload)
		fbWriteValueToWord(iValue := 0, iStartBit := 0, iEndBit := 7, wDataWord := awBusDataToVTEM[1]); 						// AddressedTargetType = 0
		fbWriteValueToWord(iValue := iMalfunctionListEntry, iStartBit := 8, iEndBit := 15, wDataWord := awBusDataToVTEM[1]);	// Index = MalfunctionListEntry
		
		awBusDataToVTEM[2] := 0; 																								// TransferValue = 0 (no value set in upload)

	4: 	// exit transfer mode
		fbWriteValueToWord(iValue := 63, iStartBit := 0, iEndBit := 5, wDataWord := awBusDataToVTEM[0]); 						// ValveMode = 63
		fbWriteValueToWord(iValue := 0, iStartBit := 6, iEndBit := 7, wDataWord := awBusDataToVTEM[0]); 						// (empty)
		fbWriteValueToWord(iValue := 0, iStartBit := 8, iEndBit := 12, wDataWord := awBusDataToVTEM[0]); 						// Channel = 0
		fbWriteValueToWord(iValue := 3, iStartBit := 13, iEndBit := 15, wDataWord := awBusDataToVTEM[0]); 						// TransferCtrl = 3 (exit)
		
		awBusDataToVTEM[1] := 0; 																								// (empty)
		awBusDataToVTEM[2] := 0; 																								// (empty)
                                                                                                            			
	5: 	// Acknowledge-Command                                                                              			
		fbWriteValueToWord(iValue := 62, iStartBit := 0, iEndBit := 5, wDataWord := awBusDataToVTEM[0]); 						// ValveMode = 62
		fbWriteValueToWord(iValue := 0, iStartBit := 6, iEndBit := 15, wDataWord := awBusDataToVTEM[0]); 						// (empty)
		awBusDataToVTEM[1] := 0; 																								// (empty)
		awBusDataToVTEM[2] := 0;		
END_CASE

END_FUNCTION_BLOCK

// auxiliary Functions/FB_Write_Value_To_Word
/// Auxiliary function block to write a value into a certain section of the data WORD 
///	The value to be written is inserted at the input iValue. 
/// The value is written from iStartBit to iEndbit.
/// The data WORD the value is written to is inserted as in-out-variable. 
/// Thereby it is possible to call the function multiple times to write into different sections of the WORD. 

FUNCTION_BLOCK FB_Write_Value_To_Word
VAR_INPUT
	iValue 		: INT; 		(* the value to be written into the specified part of the data WORD *)
	iStartBit 	: INT;	 	(* first bit of the section to be written to *)
	iEndBit 	: INT; 		(* last bit of the section to be written to *)
END_VAR
VAR_IN_OUT
	wDataWord	: WORD; 	(* data of which a section is to be written *)
END_VAR; 
VAR_OUTPUT
	xError		: BOOL; 	(* if TRUE, the value couldn't be written *)
END_VAR
VAR
	iTempVar	: INT;
	i			: INT;
END_VAR

(*****************************************************************************************************

Festo SE & Co. KG, Esslingen
Copyright (c) 2018. All rights reserved.

Product:            Motion Terminal VTEM
Description:        Function block for writing a value into a certain section of a WORD

Object version:     1.00
Last change:        2017
======================================================================================================
                                       H I S T O R Y
======================================================================================================
Version:            1.00
Date:               2017
Change/Activity:    - created
Release:            3.5.7.220
Author:             HLBG
======================================================================================================

*****************************************************************************************************)

IF iStartBit = 0 AND iEndBit = 15 THEN
	// specific treatment if the complete WORD is written as once due to the sign of integer values that could be inserted
	wDataword := INT_TO_WORD(iValue); 

ELSIF iValue < 0 OR iValue > (EXPT(2,(iEndBit-iStartBit+1))-1) THEN
	// The inserted value cannot be written into the defined section.
	
	xError := TRUE; 
	
ELSIF iStartBit < 0 OR iStartBit > 15 OR iEndBit < 0 OR iEndBit > 15 OR iStartBit > iEndBit THEN
	// The inserted bit section is not valid.
	
	xError := TRUE; 
	
ELSE
	xError := FALSE; 	

	// write the value into a temporary variable
	iTempVar := iValue;	
	
	FOR i := iStartBit TO iEndBit DO
		// write the last bit of the current tempVar into the specific section of the DataWord 
		CASE i OF
			// CASE structure is only necessary as it's not possible to address the bit directly via wDataWord.i  
			0:	wDataWord.0	 := INT_TO_BIT (iTempVar MOD 2);
			1:	wDataWord.1  := INT_TO_BIT (iTempVar MOD 2);		
			2:	wDataWord.2  := INT_TO_BIT (iTempVar MOD 2);	
			3:	wDataWord.3  := INT_TO_BIT (iTempVar MOD 2);	
			4:	wDataWord.4  := INT_TO_BIT (iTempVar MOD 2);	
			5:	wDataWord.5  := INT_TO_BIT (iTempVar MOD 2);
			6:	wDataWord.6  := INT_TO_BIT (iTempVar MOD 2);		
			7:	wDataWord.7  := INT_TO_BIT (iTempVar MOD 2);
			8:	wDataWord.8  := INT_TO_BIT (iTempVar MOD 2);		
			9:	wDataWord.9  := INT_TO_BIT (iTempVar MOD 2);	
			10: wDataWord.10 := INT_TO_BIT (iTempVar MOD 2);	
			11: wDataWord.11 := INT_TO_BIT (iTempVar MOD 2);	
			12: wDataWord.12 := INT_TO_BIT (iTempVar MOD 2);
			13: wDataWord.13 := INT_TO_BIT (iTempVar MOD 2);		
			14: wDataWord.14 := INT_TO_BIT (iTempVar MOD 2);
			15: wDataWord.15 := INT_TO_BIT (iTempVar MOD 2);		
		END_CASE
		
		// delete the last bit of the temporary variable
		iTempVar := ( iTempVar - (iTempVar MOD 2)) / 2; 		
	END_FOR
END_IF

END_FUNCTION_BLOCK

// auxiliary Functions/FB_Read_Bits_From_Word
/// Auxiliary function block to extract partial values from a value of the data type WORD.  
///	The WORD to be analysed is inserted at the input wData. 
/// The bits from iStartBit to iEndbit are analysed. Their value is the output of the function. 

FUNCTION_BLOCK FB_Read_Bits_From_Word

VAR_INPUT
	wData 		: WORD;		(* data of which a section shall be read *)
	iStartBit	: INT;		(* first bit of the section of interest *)
	iEndBit		: INT;		(* last bit of the section of interest *)
END_VAR
VAR_OUTPUT
	iValue		: INT; 		(* the value that was read *)
	xError		: BOOL; 	(* indicates if the value could be read *)
END_VAR
VAR
	i 			: INT;
	xBit 		: BOOL;
END_VAR

(*****************************************************************************************************

Festo SE & Co. KG, Esslingen
Copyright (c) 2018. All rights reserved.

Product:            Motion Terminal VTEM
Description:        Function block for reading a value out of a certain section of a WORD

Object version:     1.00
Last change:        2017
======================================================================================================
                                       H I S T O R Y
======================================================================================================
Version:            1.00
Date:               2017
Change/Activity:    - created
Release:            3.5.7.220
Author:             HLBG
======================================================================================================

*****************************************************************************************************)

IF iStartBit < 0 OR iStartBit > 15 OR iEndBit < 0 OR iEndBit > 15 OR iStartBit > iEndBit THEN
	// the start or end bit exceeds the limits of the WORD
	iValue := 0;
	xError := TRUE;
  
ELSIF iStartBit = 0 AND iEndBit = 15 THEN
	// specific treatment if the complete word is written as once due to the sign of integer values that could be inserted
	iValue := WORD_TO_INT(wData); 
	xError := FALSE; 
	
ELSE
	xError := FALSE; 
	iValue := 0 ; 
	
	FOR i := iStartBit TO iEndBit DO
	
		// read the value of a certain bit 
		CASE i OF
			// CASE structure is only necessary as it's not possible to adress the bit directly via wData.i  
			0: xBit := wData.0;
			1: xBit := wData.1;
			2: xBit := wData.2;
			3: xBit := wData.3;
			4: xBit := wData.4;
			5: xBit := wData.5;
			6: xBit := wData.6;
			7: xBit := wData.7;
			8: xBit := wData.8;
			9: xBit := wData.9;
			10: xBit := wData.10;
			11: xBit := wData.11;
			12: xBit := wData.12;
			13: xBit := wData.13;
			14: xBit := wData.14;
			15: xBit := wData.15;
		END_CASE
		
		// add the bit to the value at the correct position
		iValue := iValue + LREAL_TO_INT(BOOL_TO_INT(xBit) * EXPT(2,(i-iStartBit))); 
	END_FOR
	
END_IF

END_FUNCTION_BLOCK

// auxiliary Functions/FB_Read_Bits_From_Byte
/// Auxiliary function block to extract partial values from a value of the data type BYTE.
///	The BYTE to be analysed is inserted at the input byData.
/// The bits from iStartBit to iEndbit are analysed. Their value is the output of the function.


FUNCTION_BLOCK FB_Read_Bits_From_Byte
VAR_INPUT
	byData 		: BYTE;			(* data of which a section shall be read *)
	iStartBit	: INT;			(* first bit of the section of interest *)
	iEndBit		: INT;			(* last bit of the section of interest *)
END_VAR
VAR_OUTPUT
	byValue		: BYTE; 		(* the value that was read *)
	xError		: BOOL; 		(* indicates if the value could be read *)
END_VAR
VAR
	i 			: INT;
	xBit 		: BOOL;
END_VAR

(*****************************************************************************************************

Festo SE & Co. KG, Esslingen
Copyright (c) 2018. All rights reserved.

Product:            Motion Terminal VTEM
Description:        Function block for reading a value out of a certain section of a BYTE

Object version:     1.00
Last change:        2017
======================================================================================================
                                       H I S T O R Y
======================================================================================================
Version:            1.00
Date:               2017
Change/Activity:    - created
Release:            3.5.7.220
Author:             HLBG
======================================================================================================

*****************************************************************************************************)

IF iStartBit < 0 OR iStartBit > 7 OR iEndBit < 0 OR iEndBit > 7 OR iStartBit > iEndBit THEN
	// the start or end bit exceeds the limits of the BYTE
	byValue := 0;
	xError := TRUE;
  
ELSE
	xError := FALSE; 
	byValue := 0; 
	
	FOR i := iStartBit TO iEndBit DO
	
		// read the value of a specific bit
		CASE i OF
			// CASE structure is only necessary as it's not possible to address the bit directly via byData.i  
			0: xBit := byData.0;
			1: xBit := byData.1;
			2: xBit := byData.2;
			3: xBit := byData.3;
			4: xBit := byData.4;
			5: xBit := byData.5;
			6: xBit := byData.6;		
			7: xBit := byData.7;
		END_CASE
		
		// add the bit to the value at the correct position
		byValue := byValue + LREAL_TO_BYTE(BOOL_TO_BYTE(xBit) * EXPT(2,(i-iStartBit)));
	END_FOR
	
END_IF

END_FUNCTION_BLOCK

// StateInterpreter/FB_StateInterpreter_MA_01
/// The variable "byActualAppState" is an output of the FB_ValveControl that is used differently in each Motion App.
/// This function block interprets the "AppState" output of the FB_ValveControl if Motion App 1 ("Directional control valve functions") is running.
/// The Motion App specific values are derived from the "byActualAppState".

FUNCTION_BLOCK FB_StateInterpreter_MA_01
VAR_INPUT
	byActualAppState 			: BYTE; 	(* output of the FB_ValveControl *)
END_VAR
VAR_OUTPUT
	xRetractedEndPos_optional	: BOOL;  	(* only if digital sensors are installed (optional): indicates whether the retracted end position was reached (after outlet port 2 is pressurised) *)
	xAdvancedEndPos_optional	: BOOL;  	(* only if digital sensors are installed (optional): indicates whether the advanced end position was reached (after outlet port 4 is pressurised) *)
	bySwitchingPositionAt2 		: BYTE;  	(* indicates the switching position at outlet port 2 *)
	bySwitchingPositionAt4 		: BYTE;		(* indicates the switching position at outlet port 4 *)
	xWarning					: BOOL; 	(* indicates whether there is a warning returned by the Motion App *)
END_VAR
VAR
	fbReadBitsFromByte		: FB_Read_Bits_From_Byte;
	byRetractedEndPos		: BYTE;
	byAdvancedEndPos		: BYTE;
	byWarning				: BYTE;
END_VAR

(*****************************************************************************************************

Festo SE & Co. KG, Esslingen
Copyright (c) 2018. All rights reserved.

Product:            Motion Terminal VTEM
Description:        Function block for interpreting the app state of Motion App 1

Object version:     1.00
Last change:        2017
======================================================================================================
                                       H I S T O R Y
======================================================================================================
Version:            1.00
Date:               2017
Change/Activity:    - created
Release:            3.5.7.220
Author:             HLBG
======================================================================================================

*****************************************************************************************************)

// read the Motion App specific values from the ActualAppState byte
fbReadBitsFromByte(byData := byActualAppState, iStartBit := 0, iEndBit := 0, byValue => byRetractedEndPos);
xRetractedEndPos_optional :=  BYTE_TO_BIT(byRetractedEndPos);

fbReadBitsFromByte(byData := byActualAppState, iStartBit := 2, iEndBit := 2, byValue => byAdvancedEndPos); 
xAdvancedEndPos_optional :=  BYTE_TO_BIT(byAdvancedEndPos);

fbReadBitsFromByte(byData := byActualAppState, iStartBit := 3, iEndBit := 4, byValue => bySwitchingPositionAt2);

fbReadBitsFromByte(byData := byActualAppState, iStartBit := 5, iEndBit := 6, byValue => bySwitchingPositionAt4);

fbReadBitsFromByte(byData := byActualAppState, iStartBit := 7, iEndBit := 7, byValue => byWarning);
xWarning := BYTE_TO_BIT(byWarning);

END_FUNCTION_BLOCK

// StateInterpreter/FB_StateInterpreter_MA_11
/// The variable "byActualAppState" is an output of the FB_ValveControl that is used differently in each Motion App.
/// This function block interprets the "AppState" output of the FB_ValveControl if Motion App 11 ("Soft stop") is running.
/// The Motion App specific values are derived from the "byActualAppState".

FUNCTION_BLOCK FB_StateInterpreter_MA_11
VAR_INPUT
	byActualAppState 		: BYTE; 	(* output of the FB_ValveControl *)
END_VAR
VAR_OUTPUT
	xRetractedEndPos		: BOOL;  	(* indicates whether the retracted end position was reached (after outlet port 2 is pressurised) *)
	xAdvancedEndPos			: BOOL;  	(* indicates whether the advanced end position was reached (after outlet port 4 is pressurised) *)
	xContactPressure		: BOOL;		(* indicates whether the internal calculated contact pressure was reached *)
	xPistonDetectRet		: BOOL;		// indicates whether the piston is detected within the sensing range of the sensor at the retracted end position
	xPistonDetectAdv		: BOOL;		// indicates whether the piston is detected within the sensing range of the sensor at the advanced end position
	xWarning				: BOOL; 	(* indicates whether there is a warning returned by the Motion App *)
END_VAR
VAR
	fbReadBitsFromByte		: FB_Read_Bits_From_Byte;
	byRetractedEndPos		: BYTE;
	byAdvancedEndPos		: BYTE;
	byPistonDetectRet		: BYTE;
	byPistonDetectAdv		: BYTE;
	byWarning				: BYTE;
	byContactPressure		: BYTE;
END_VAR

(*****************************************************************************************************

Festo SE & Co. KG, Esslingen
Copyright (c) 2018. All rights reserved.

Product:            Motion Terminal VTEM
Description:        Function block for interpreting the app state of Motion App 11 

Object version:     1.02
Last change:        2018-11
======================================================================================================
                                       H I S T O R Y
======================================================================================================
Version:            1.02
Date:               2018-11
Change/Activity:    - added outputs xPistonDetectRet and xPistonDetectAdv (#2248541)
Release:            3.5.7.222
Author:             JEBU
------------------------------------------------------------------------------------------------------
Version:            1.01
Date:               2018-08
Change/Activity:    - added output xContactPressure (#2257121)
Release:            3.5.7.220
Author:             JEBU
------------------------------------------------------------------------------------------------------
Version:            1.00
Date:               2017
Change/Activity:    - created
Release:            3.5.7.220
Author:             HLBG
======================================================================================================

*****************************************************************************************************)

// read the Motion App specific values from the ActualAppState byte
fbReadBitsFromByte(byData := byActualAppState, iStartBit := 0, iEndBit := 0, byValue => byRetractedEndPos);
xRetractedEndPos :=  BYTE_TO_BIT(byRetractedEndPos);

fbReadBitsFromByte(byData := byActualAppState, iStartBit := 1, iEndBit := 1, byValue => byContactPressure);
xContactPressure := BYTE_TO_BIT(byContactPressure);

fbReadBitsFromByte(byData := byActualAppState, iStartBit := 2, iEndBit := 2, byValue => byAdvancedEndPos);
xAdvancedEndPos :=  BYTE_TO_BIT(byAdvancedEndPos);

fbReadBitsFromByte(byData := byActualAppState, iStartBit := 3, iEndBit := 3, byValue => byPistonDetectRet);
xPistonDetectRet :=  BYTE_TO_BIT(byPistonDetectRet);

fbReadBitsFromByte(byData := byActualAppState, iStartBit := 4, iEndBit := 4, byValue => byPistonDetectAdv);
xPistonDetectAdv :=  BYTE_TO_BIT(byPistonDetectAdv);

fbReadBitsFromByte(byData := byActualAppState, iStartBit := 7, iEndBit := 7, byValue => byWarning);
xWarning := BYTE_TO_BIT(byWarning);

END_FUNCTION_BLOCK

// StateInterpreter/FB_StateInterpreter_MA_12
/// The variable "byActualAppState" is an output of the FB_ValveControl that is used differently in each Motion App.
/// This function block interprets the "AppState" output of the FB_ValveControl if Motion App 12 ("Leakage diagnostics") is running.
/// The Motion App specific values are derived from the "byActualAppState".

FUNCTION_BLOCK FB_StateInterpreter_MA_12
VAR_INPUT
	byActualAppState 		: BYTE; 	(* output of the FB_ValveControl *)
END_VAR
VAR_OUTPUT
	byStateLeakageAt2 		: BYTE;  	(* evaluates the measured leakage increase at outlet port 2 (0 = defect/failure, 1 = critical, 2 = warning, 3 = good) *)
	byStateLeakageAt4 		: BYTE;  	(* evaluates the measured leakage increase at outlet port 4 (0 = defect/failure, 1 = critical, 2 = warning, 3 = good) *)
	byStateProcedure 		: BYTE;  	(* indicates the state of the leakage-measurement-procedure *)
	xWarning				: BOOL; 	(* indicates whether there is a warning returned by the Motion App *)
END_VAR
VAR
	fbReadBitsFromByte		: FB_Read_Bits_From_Byte;
	byWarning				: BYTE;
END_VAR

(*****************************************************************************************************

Festo SE & Co. KG, Esslingen
Copyright (c) 2018. All rights reserved.

Product:            Motion Terminal VTEM
Description:        Function block for interpreting the app state of Motion App 12 

Object version:     1.00
Last change:        2017
======================================================================================================
                                       H I S T O R Y
======================================================================================================
Version:            1.00
Date:               2017
Change/Activity:    - created
Release:            3.5.7.220
Author:             HLBG
======================================================================================================

*****************************************************************************************************)

// read the Motion App specific values from the ActualAppState byte
fbReadBitsFromByte(byData := byActualAppState, iStartBit := 0, iEndBit := 1, byValue => byStateLeakageAt2);

fbReadBitsFromByte(byData := byActualAppState, iStartBit := 2, iEndBit := 3, byValue => byStateLeakageAt4);

fbReadBitsFromByte(byData := byActualAppState, iStartBit := 4, iEndBit := 6, byValue => byStateProcedure);

fbReadBitsFromByte(byData := byActualAppState, iStartBit := 7, iEndBit := 7, byValue => byWarning);
xWarning := BYTE_TO_BIT(byWarning);

END_FUNCTION_BLOCK

// StateInterpreter/FB_StateInterpreter_MA_06
/// The variable "byActualAppState" is an output of the FB_ValveControl that is used differently in each Motion App.
/// This function block interprets the "AppState" output of the FB_ValveControl if Motion App 6 ("ECO drive") is running.
/// The Motion App specific values are derived from the "byActualAppState".

FUNCTION_BLOCK FB_StateInterpreter_MA_06
VAR_INPUT
	byActualAppState 		: BYTE; 	(* output of the FB_ValveControl *)
END_VAR
VAR_OUTPUT
	xRetractedEndPos		: BOOL;  	(* indicates whether the retracted end position was reached (after outlet port 2 is pressurised) *)
	xAdvancedEndPos			: BOOL;  	(* indicates whether the advanced end position was reached (after outlet port 4 is pressurised) *)
	xWarning				: BOOL; 	(* indicates whether there is a warning returned by the Motion App *)
END_VAR
VAR
	fbReadBitsFromByte		: FB_Read_Bits_From_Byte;
	byRetractedEndPos		: BYTE;
	byAdvancedEndPos		: BYTE;
	byWarning				: BYTE;
END_VAR

(*****************************************************************************************************

Festo SE & Co. KG, Esslingen
Copyright (c) 2018. All rights reserved.

Product:            Motion Terminal VTEM
Description:        Function block for interpreting the app state of Motion App 6

Object version:     1.00
Last change:        2017
======================================================================================================
                                       H I S T O R Y
======================================================================================================
Version:            1.00
Date:               2017
Change/Activity:    - created
Release:            3.5.7.220
Author:             HLBG
======================================================================================================

*****************************************************************************************************)

// read the Motion App specific values from the ActualAppState byte
fbReadBitsFromByte(byData := byActualAppState, iStartBit := 0, iEndBit := 0, byValue => byRetractedEndPos);
xRetractedEndPos :=  BYTE_TO_BIT(byRetractedEndPos);

fbReadBitsFromByte(byData := byActualAppState, iStartBit := 2, iEndBit := 2, byValue => byAdvancedEndPos); 
xAdvancedEndPos :=  BYTE_TO_BIT(byAdvancedEndPos);

fbReadBitsFromByte(byData := byActualAppState, iStartBit := 7, iEndBit := 7, byValue => byWarning);
xWarning := BYTE_TO_BIT(byWarning);

END_FUNCTION_BLOCK

// Transfermode/specific_MA_config/FB_Write_config_MA_07
/// This function block can be used to download the configuration of Motion App 7 ("Presetting of travel time").
/// The specific parameters of this Motion App are the inputs of this FB and can be defined by the user. 
/// The function block uses the transfer mode to write this configuration to the Motion Terminal
/// and indicates the state of the download process.

FUNCTION_BLOCK FB_Write_config_MA_07
VAR_INPUT
	awBusDataFromVTEM 				: ARRAY [0..2] OF WORD;		(* 6 bytes of process data received from the Motion Terminal *)
END_VAR

VAR_IN_OUT
	awBusDataToVTEM 				: ARRAY [0..2] OF WORD; 	(* 6 bytes of process data sent to the Motion Terminal *)
END_VAR

VAR_INPUT
	xExecute 						: BOOL; 					(* has to be set to TRUE for a download and to FALSE to reset the function block after a download *)
		                    		                        	
	iParameterSet					: INT := 1; 				(* the parameter set to be written to, 1 by default *)
	
	// system parameters                 		                        	
		iTubingLengthAt2 			: INT; 						(* length of the tubing connected to outlet port 2 of the valve [1 digit = 1 mm] *)
 		iTubingLengthAt4 			: INT;						(* length of the tubing connected to outlet port 4 of the valve [1 digit = 1 mm] *)
 		iTubingInnerDiameterAt2		: INT;  					(* inner diameter of the tubing connected to outlet port 2 of the valve [1 digit = 0.01 mm] *)
 		iTubingInnerDiameterAt4		: INT;						(* inner diameter of the tubing connected to outlet port 4 of the valve [1 digit = 0.01 mm] *)
 		iDriveType 					: INT;						(* type of the drive/cylinder/... that is to be operated by the valve ->  see list of drive types *)
 		iDriveStroke 				: INT; 						(* stroke of the drive/cylinder/... that is to be operated by the valve [1 digit = 1 mm for linear drives, 1 digit = 1° for rotary drives] *)
		iInstallationPositionDrive 	: INT;  	 				(* inclination of the cylinder with reference to a horizontal installation position [1 digit = 0.01°, positive values = advancing upwards] *)
		iInPortRetracted			: INT;						// Sensor port for detection of end position at pressurisation of outlet port 2 (retracted), value is number of the slot (beginning from 0) * 10 + number of the port
		iInPortAdvanced				: INT;						// Sensor port for detection of end position at pressurisation of outlet port 4 (advanced), value is number of the slot (beginning from 0) * 10 + number of the port
	                                                        	
	// application parameters                               	
		iLoadRetracting 			: INT;						(* mass that is to be moved by the drive when retracting ((2) pressurised) [1 digit = 0.01 kg] *)
 		iLoadAdvancing 				: INT; 						(* mass that is to be moved by the drive when advancing ((4) pressurised) [1 digit = 0.01 kg] *)
		iMomentOfInertiaRetracting	: INT;						// Moment of inertia during for swivel drives when retratcting ((2) pressirised) [1 digit = 1 kg cm³]
		iMomentOfInertiaAdvancing	: INT;						// Moment of inertia during for swivel drives when advancing ((4) pressirised) [1 digit = 1 kg cm³]
		iTravelTimeRetracting 		: INT;						(* preset travel time from one end position to the other when retracting ((2) pressurised) [1 digit = 0.01 s] *)
		iTravelTimeAdvancing 		: INT; 						(* preset travel time from one end position to the other when advancing ((4) pressurised) [1 digit = 0.01 s] *)
		iSoftStartFunction			: INT := 1;					(* flag to enable or disable the iSoftStartFunction; 0 = disabled, 1 = enabled *)
END_VAR

VAR_OUTPUT                                                  	
	iResponse 						: eTransferResponse; 		(* returns the status of the execution of the download process *)
	sCurrentValue 					: STRING; 					(* indicates which value of the array is currently treated (necessary to evaluate in case of error messages) *)
	xDownloadDone 					: BOOL; 					(* indicates whether the download was successful *)
	xDownloadError 					: BOOL := FALSE; 			(* indicates whether an error occurred during the transfer *)
END_VAR

VAR
	aTransferPackages				: ARRAY [0..100] OF stTransferPackage;
	fbdownloadMultipleParameters 	: FB_Download_Multiple_Parameters;
	iCurrentValue					: INT;
	fbWriteValueToWord 				: FB_Write_Value_To_Word;
END_VAR

(*****************************************************************************************************

Festo SE & Co. KG, Esslingen
Copyright (c) 2018. All rights reserved.

Product:            Motion Terminal VTEM
Description:        Function block to download the parameters for Motion App 7 to the Motion Terminal

Object version:     2.00
Last change:        2019-03
======================================================================================================
                                       H I S T O R Y
======================================================================================================
Version:            2.00
Date:               2019-03
Change/Activity:    - added parameters for moment of inertia used for swivel drives (#2307852)
                    - added parameters for the sensor port mapping (#2256294)
                    - changed awBusDataToVTEM into VAR_IN_OUT (#2368965)
Release:            3.5.7.230 (CODESYS 3.5.7.2, Lib version 3.0)
Author:             JEBU
------------------------------------------------------------------------------------------------------
Version:            1.00
Date:               2017
Change/Activity:    - created
Release:            3.5.7.220
Author:             HLBG
======================================================================================================

*****************************************************************************************************)

// write the Motion App specific parameters into the struct
	//iTubingLengthAt2
		aTransferPackages[0].iChannel := iParameterSet;
		aTransferPackages[0].iAddressedTarget := 7;
		aTransferPackages[0].iIndex := 12;
		aTransferPackages[0].iTransferValue := iTubingLengthAt2;
		
	//iTubingLengthAt4
		aTransferPackages[1].iChannel := iParameterSet;
		aTransferPackages[1].iAddressedTarget := 7;
		aTransferPackages[1].iIndex := 13;
		aTransferPackages[1].iTransferValue := iTubingLengthAt4;
		
	//iTubingInnerDiameterAt2
		aTransferPackages[2].iChannel := iParameterSet;
		aTransferPackages[2].iAddressedTarget := 7;
		aTransferPackages[2].iIndex := 14;
		aTransferPackages[2].iTransferValue := iTubingInnerDiameterAt2;
		
	//iTubingInnerDiameterAt4
		aTransferPackages[3].iChannel := iParameterSet;
		aTransferPackages[3].iAddressedTarget := 7;
		aTransferPackages[3].iIndex := 15;
		aTransferPackages[3].iTransferValue := iTubingInnerDiameterAt4;
		
	//iDriveType
		aTransferPackages[4].iChannel := iParameterSet;
		aTransferPackages[4].iAddressedTarget := 7;
		aTransferPackages[4].iIndex := 20;
		aTransferPackages[4].iTransferValue := iDriveType;
		
	//iDriveStroke
		aTransferPackages[5].iChannel := iParameterSet;
		aTransferPackages[5].iAddressedTarget := 7;
		aTransferPackages[5].iIndex := 21;
		aTransferPackages[5].iTransferValue := iDriveStroke;
		
	//iInstallationPositionDrive
		aTransferPackages[6].iChannel := iParameterSet;
		aTransferPackages[6].iAddressedTarget := 7;
		aTransferPackages[6].iIndex := 60;
		aTransferPackages[6].iTransferValue := iInstallationPositionDrive;
		
	//iLoadRetracting
		aTransferPackages[7].iChannel := iParameterSet;
		aTransferPackages[7].iAddressedTarget := 7;
		aTransferPackages[7].iIndex := 100;
		aTransferPackages[7].iTransferValue := iLoadRetracting;
		
	//iLoadAdvancing
		aTransferPackages[8].iChannel := iParameterSet;
		aTransferPackages[8].iAddressedTarget := 7;
		aTransferPackages[8].iIndex := 101;
		aTransferPackages[8].iTransferValue := iLoadAdvancing;
		
	//iMomentOfInertiaRetracting
		aTransferPackages[9].iChannel := iParameterSet;
		aTransferPackages[9].iAddressedTarget := 7;
		aTransferPackages[9].iIndex := 102;
		aTransferPackages[9].iTransferValue := iMomentOfInertiaRetracting;
	
	//iMomentOfInertiaAdvancing
		aTransferPackages[10].iChannel := iParameterSet;
		aTransferPackages[10].iAddressedTarget := 7;
		aTransferPackages[10].iIndex := 103;
		aTransferPackages[10].iTransferValue := iMomentOfInertiaAdvancing;

	//iTravelTimeRetracting
		aTransferPackages[11].iChannel := iParameterSet;
		aTransferPackages[11].iAddressedTarget := 7;
		aTransferPackages[11].iIndex := 120;
		aTransferPackages[11].iTransferValue := iTravelTimeRetracting;
	
	//iTravelTimeAdvancing
		aTransferPackages[12].iChannel := iParameterSet;
		aTransferPackages[12].iAddressedTarget := 7;
		aTransferPackages[12].iIndex := 121;
		aTransferPackages[12].iTransferValue := iTravelTimeAdvancing;
	
	//iSoftStartFunction
		aTransferPackages[13].iChannel := iParameterSet;
		aTransferPackages[13].iAddressedTarget := 7;
		aTransferPackages[13].iIndex := 222;
		aTransferPackages[13].iTransferValue := iSoftStartFunction;
	
	//iInPortRetract
		aTransferPackages[14].iChannel := iParameterSet;
		aTransferPackages[14].iAddressedTarget := 7;
		aTransferPackages[14].iIndex := 70;
		aTransferPackages[14].iTransferValue := iInPortRetracted;
	
	//iInPortRetract
		aTransferPackages[15].iChannel := iParameterSet;
		aTransferPackages[15].iAddressedTarget := 7;
		aTransferPackages[15].iIndex := 71;
		aTransferPackages[15].iTransferValue := iInPortAdvanced;
	
	// define end of parameter list to be downloaded by setting all variables to 0 (end criterion for FB_Download_Multiple_Parameters)
		aTransferPackages[16].iChannel := 0;
		aTransferPackages[16].iAddressedTarget := 0;
		aTransferPackages[16].iIndex := 0;
		aTransferPackages[16].iTransferValue := 0;


// pre-check of the value for the parameter set
	IF xExecute = TRUE AND (iParameterSet < 1 OR iParameterSet > 5) THEN		// invalid input for the parameter set
		xDownloadDone := FALSE; 
		xDownloadError := TRUE; 
		iResponse := eTransferResponse.invalid_ParameterSet; 
		iCurrentValue := 0; 
		// send command 'stop'
		fbWriteValueToWord(iValue := 61, iStartBit := 0, iEndBit := 5, wDataWord := awBusDataToVTEM[0]); 			// ValveMode = 61
		fbWriteValueToWord(iValue := 0, iStartBit := 6, iEndBit := 15, wDataWord := awBusDataToVTEM[0]); 			// (empty)
		awBusDataToVTEM[1] := 0; 
		awBusDataToVTEM[2] := 0; 
		
	ELSE	
		// call the function block for multiple parameter download
			fbdownloadMultipleParameters(	xExecute := xExecute,
											awBusDataFromVTEM := awBusDataFromVTEM,
											aTransferPackages := aTransferPackages, 
											awBusDataToVTEM := awBusDataToVTEM,
											xDownloadDone => xDownloadDone,
											xDownloadError => xDownloadError,
											iResponse => iResponse,
											iCurrentValue => iCurrentValue);
	END_IF


// The current value output is needed if there is any invalid value in order to address it correctly.
// As the user doesn't work with indices in this function block, the current value is transformed to a string holding the name of the parameter.
	CASE iCurrentValue OF
		0: sCurrentValue := 'iTubingLengthAt2';
		1: sCurrentValue := 'iTubingLengthAt4';
		2: sCurrentValue := 'iTubingInnerDiameterAt2';
		3: sCurrentValue := 'iTubingInnerDiameterAt4';
		4: sCurrentValue := 'iDriveType';
		5: sCurrentValue := 'iDriveStroke';
		6: sCurrentValue := 'iInstallationPositionDrive';
		7: sCurrentValue := 'iLoadRetracting';
		8: sCurrentValue := 'iLoadAdvancing';
		9: sCurrentValue := 'iMomentOfInertiaRetracting';
		10: sCurrentValue := 'iMomentOfInertiaAdvancing';
		11: sCurrentValue := 'iTravelTimeRetracting';
		12: sCurrentValue := 'iTravelTimeAdvancing';
		13: sCurrentValue := 'iSoftStartFunction';
		14: sCurrentValue := 'iInPortRetract';
		15: sCurrentValue := 'iInPortAdvanced';
		16: sCurrentValue := 'AllParametersWritten';
	END_CASE

END_FUNCTION_BLOCK

// Transfermode/FB_Download_Multiple_Parameters
/// This function block can be used to run the transfer mode of the Motion Terminal in order to download multiple values.
/// The values to be downloaded are handed over as a structured list, indicating the channel, the addressed target and the index of each value.

FUNCTION_BLOCK FB_Download_Multiple_Parameters
VAR_INPUT
	awBusDataFromVTEM 		: ARRAY [0..2] OF WORD; 				(* 6 bytes of process data received from the Motion Terminal *)
END_VAR	

VAR_IN_OUT
	awBusDataToVTEM 		: ARRAY [0..2] OF WORD; 				(* 6 bytes of process data sent to the Motion Terminal *)
END_VAR

VAR_INPUT
	xExecute 				: BOOL; 								(* has to be set to TRUE for a download and to FALSE to reset the function block after a download *)
	aTransferPackages 		: ARRAY [0..100] OF stTransferPackage;	(* array that is used to address and specify the values to be downloaded *)
END_VAR

VAR_OUTPUT
	iResponse 				: eTransferResponse; 					(* returns the status of the execution of the download process *)
	iCurrentValue 			: INT; 									(* indicates which array index is currently treated (necessary to evaluate in case of error messages) *)
	xDownloadDone 			: BOOL; 								(* indicates whether the download was successful *)
	xDownloadError 			: BOOL; 								(* indicates whether an error occurred during the transfer *)
END_VAR

VAR
	iRecValveMode 			: INT;
	iRecValveStatus 		: eValveState;
	iCommandNumber			: INT; 									(* indicates the command to be executed *)
	fbWriteValueToWord		: FB_Write_Value_To_Word;
	fbReadBitsFromWord 		: FB_Read_Bits_From_Word;
	iRecChannel				: INT;
	iRecTransferCtrl		: INT;
	iRecAddressedTargetType	: INT;
	iRecIndex				: INT;
	iRecTransferValue		: INT;
	
	iAppStatus				: INT;
	xFirstCycle				: BOOL := TRUE;
	xTransferComplete		: BOOL;
	aFCTransferPackages		: ARRAY [0..100] OF stTransferPackage;
	iLength					: INT;
	i						: INT;
	xInputValid				: BOOL;
	xInputConsistent		: BOOL;
	iFCLength				: INT;
	xStopPending			: BOOL;
END_VAR

(*****************************************************************************************************

Festo SE & Co. KG, Esslingen
Copyright (c) 2018. All rights reserved.

Product:            Motion Terminal VTEM
Description:        Function block to download multiple parameters to the Motion Terminal

Object version:     2.01
Last change:        2019-07
======================================================================================================
                                       H I S T O R Y
======================================================================================================
Version:            2.01 
Date:               2019-07        
Change/Activity:    - adjusted range for iChannel from 255 to 31 (#2510540)
					- validity check shows first wrong element and stops the procedure (#2526112)
					- adapted functionality for transfer mode on slots without valves (#2957509)
					- added new enum value (#3104444)
Release:            3.5.7.234 (CODESYS 3.5.7.2, Lib version 3.4)
Author:             MKLP/JEBU
------------------------------------------------------------------------------------------------------
Version:            2.00
Date:               2019-03
Change/Activity:    - changed awBusDataToVTEM into VAR_IN_OUT (#2368965)
                    - fixed bug that caused "exit transfer mode" even if xExecute is FALSE (#2181575)
                    - added value 7 to list of invalid commands (#2318899)
Release:            3.5.7.230 (CODESYS 3.5.7.2, Lib version 3.0)
Author:             JEBU/MKLP
------------------------------------------------------------------------------------------------------
Version:            1.01
Date:               2018-11
Change/Activity:    - adjusted value range of iChannel and iAddressedTarget to 0...255 (#2181575)
Release:            3.5.7.221 (CODESYS 3.5.7.2, Lib version 2.1)
Author:             JEBU
------------------------------------------------------------------------------------------------------
Version:            1.00
Date:               2017
Change/Activity:    - created
Release:            3.5.7.22 (CODESYS 3.5.7.2, Lib version 2.0)
Author:             HLBG
======================================================================================================

*****************************************************************************************************)

// read the ValveMode and the ValveState of the Motion Terminal
fbReadBitsFromWord(wData := awBusDataFromVTEM[0], iStartBit := 0, iEndBit := 5, iValue => iRecValveMode);
fbReadBitsFromWord(wData := awBusDataFromVTEM[0], iStartBit := 6, iEndBit := 7, iValue => iRecValveStatus);

// A rising edge at xExecute indicates that new values are to be written, xExecute must be TRUE during the whole download procedure
IF xExecute = TRUE THEN	
	// pre-analysis of the input data before caring about the transfer
	IF xFirstCycle = TRUE THEN
		// reset StopPending	
		xStopPending := FALSE;
		
		// store the parameter array that was given in the first cycle
		aFCTransferPackages := aTransferPackages;

		// get the length of the parameter array
		iLength := 0; 
		WHILE (aTransferPackages [iLength].iChannel <> 0 OR aTransferPackages [iLength].iAddressedTarget <> 0 OR aTransferPackages [iLength].iIndex <> 0 OR aTransferPackages [iLength].iTransferValue <> 0) DO
			iLength := iLength + 1; 
		END_WHILE
		iFCLength := iLength;
				
		// check the single data items of the array
		xInputValid := TRUE;
		xInputConsistent := TRUE;
			
		FOR i := 0 TO iLength DO
			IF aTransferPackages [i].iChannel < 0 OR aTransferPackages [i].iChannel > 31 THEN
				iResponse := eTransferResponse.invalid_Channel;
				iCurrentValue := i;
				xInputValid := FALSE;
				EXIT;
			ELSIF aTransferPackages [i].iAddressedTarget < 0 OR aTransferPackages [i].iAddressedTarget > 255 THEN
				iResponse := eTransferResponse.invalid_AddressedTarget;
				iCurrentValue := i;
				xInputValid := FALSE;
				EXIT;
			ELSIF aTransferPackages[i].iIndex < 0 OR aTransferPackages[i].iIndex > 255 THEN
				iResponse := eTransferResponse.invalid_Index;
				iCurrentValue := i;
				xInputValid := FALSE;
				EXIT;
			END_IF
		END_FOR
		
	ELSE	// xFirstCycle = FALSE
		// check whether the current command is still the same compared to the command at the rising edge of xExecute
		
		// get the length of the parameter array
		iLength := 0; 
		WHILE (aTransferPackages[iLength].iChannel <> 0 OR aTransferPackages[iLength].iAddressedTarget <> 0 OR aTransferPackages[iLength].iIndex <> 0 OR aTransferPackages[iLength].iTransferValue <> 0) DO
			iLength := iLength + 1;
		END_WHILE
		
		// check length and content of the array by comparing it to the array of the first cycle
		IF iFCLength <> iLength THEN
			xInputConsistent := FALSE;
			iResponse := eTransferResponse.FB_needs_rising_edge_xExecute;
  		ELSE
			FOR i := 0 TO iLength DO
				IF aFCTransferPackages[i].iChannel <> aTransferPackages[i].iChannel THEN
					xInputConsistent := FALSE;
					iResponse := eTransferResponse.FB_needs_rising_edge_xExecute;
				ELSIF aFCTransferPackages[i].iAddressedTarget <> aTransferPackages[i].iAddressedTarget THEN
					xInputConsistent := FALSE;
					iResponse := eTransferResponse.FB_needs_rising_edge_xExecute;
				ELSIF aFCTransferPackages[i].iIndex <> aTransferPackages[i].iIndex THEN
					xInputConsistent := FALSE;
					iResponse := eTransferResponse.FB_needs_rising_edge_xExecute;
				ELSIF aFCTransferPackages[i].iTransferValue <> aTransferPackages[i].iTransferValue THEN
					xInputConsistent := FALSE;
					iResponse := eTransferResponse.FB_needs_rising_edge_xExecute;
				END_IF
			END_FOR
		END_IF
	END_IF 		// end of pre-analysis of the input data

	IF xInputConsistent = TRUE AND xInputValid = TRUE THEN
		IF iRecValveStatus = eValveState.Running THEN		// a Motion App is running
			iResponse := eTransferResponse.preparing_transfer;
			iCommandNumber := 3; 					// command 'stop'
			xDownloadError := FALSE;
			
		ELSE	// The transfer mode can be used as the ValveStatus is not RUNNING
			IF iCommandNumber = 1 THEN // If transfer started with a virtual valve, eNum will be overwritten
				iResponse := eTransferResponse.transferring;
			END_IF
			
			IF iRecValveMode <> 63 AND xDownloadDone = FALSE THEN	// The transfer mode is currently not active and the values are not downloaded yet
				// check whether the WebConfig blocks the access to transfer mode
				fbReadBitsFromWord(wData := awBusDataFromVTEM[0], iStartBit := 8, iEndBit := 15, iValue => iAppStatus);
				IF iRecValveMode = 61 AND iAppStatus = 10 THEN 		// access denied by WebConfig
					xDownloadError := TRUE;
					iResponse := eTransferResponse.access_denied_WebConfig;
					iCommandNumber := 3; 			// do nothing (here: command 'stop')
				ELSIF iRecValveMode = 61 AND iAppStatus = 11 THEN 	// access denied due to an active saving process
					xDownloadError := TRUE;
					iResponse := eTransferResponse.access_denied_saving;
					iCommandNumber := 3; 			// do nothing (here: command 'stop')
				ELSIF iRecValveMode = 61 AND iAppStatus = 15 THEN 	// no valve detected
					xDownloadError := TRUE;
					iResponse := eTransferResponse.no_valve_detected; 
					iCommandNumber := 1; 			// keep downloading (here: command 'download') In a Firmware older than 4.16(E) an empty valve keep sending ValveMode 61 and AppStatus 15. In Firmware 4.16(E) the message changes with a tranfer
				ELSIF iRecValveMode = 61 AND iAppStatus = 0 AND xTransferComplete = TRUE THEN
					// All values are downloaded and the transfer mode has been closed properly
					xDownloadDone := TRUE;
					xDownloadError := FALSE;
					iCommandNumber := 3; 			// command 'stop' to remain the valve stopped
				ELSE	// ready to start transfer mode
					xDownloadError := FALSE;
					iResponse := eTransferResponse.transferring;
					iCommandNumber := 1; 			// command 'download' for the current value
				END_IF
		
			ELSIF iRecValveMode = 63 AND xDownloadDone = FALSE THEN		// The transfer mode is active, but the values are not downloaded yet
				fbReadBitsFromWord(wData := awBusDataFromVTEM[0], iStartBit := 8, iEndBit := 12, iValue => iRecChannel);
				fbReadBitsFromWord(wData := awBusDataFromVTEM[0], iStartBit := 13, iEndBit := 15, iValue => iRecTransferCtrl);
				fbReadBitsFromWord(wData := awBusDataFromVTEM[1], iStartBit := 0, iEndBit := 7, iValue => iRecAddressedTargetType);
				fbReadBitsFromWord(wData := awBusDataFromVTEM[1], iStartBit := 8, iEndBit := 15, iValue => iRecIndex);
				iRecTransferValue := WORD_TO_INT(awBusDataFromVTEM[2]);
		 
				IF aTransferPackages[iCurrentValue].iChannel = iRecChannel AND iRecTransferCtrl = 1 AND aTransferPackages[iCurrentValue].iAddressedTarget = iRecAddressedTargetType AND
					aTransferPackages[iCurrentValue].iIndex = iRecIndex AND  aTransferPackages[iCurrentValue].iTransferValue = iRecTransferValue THEN
						// The download command for the parameter was mirrored by the Motion Terminal, the download has been confirmed
						
						xDownloadError := FALSE;
						iCurrentValue := iCurrentValue +1;		// next value
						
						// check whether there is another value
						IF aTransferPackages[iCurrentValue].iAddressedTarget = 0 AND aTransferPackages[iCurrentValue].iChannel = 0 AND aTransferPackages[iCurrentValue].iIndex = 0 AND
							aTransferPackages[iCurrentValue].iTransferValue = 0 THEN 	// last value reached
							
							iCommandNumber := 2; 		// exit transfer mode
							iResponse := eTransferResponse.transfer_successful;
							xTransferComplete := TRUE;
							xStopPending := TRUE;
						ELSE
							iCommandNumber := 1; 		// command 'download' for the (next) value
							iResponse := eTransferResponse.transferring;
						END_IF
					
				ELSIF iRecChannel = 0 AND iRecTransferCtrl = 0 AND iRecAddressedTargetType = 0 AND iRecIndex = 0 AND iRecTransferValue <> 0 AND xFirstCycle = FALSE THEN
					// An invalid command was sent when using the transfer mode
					
					iCommandNumber := 1; 			// command 'download' for the current value
					xDownloadError := TRUE; 
					
					CASE iRecTransferValue OF		// indicates the type of the invalid command
						1: 	iResponse := eTransferResponse.invalid_Channel;
						2: 	iResponse := eTransferResponse.invalid_TransferControl;	// this should never happen
						3: 	iResponse := eTransferResponse.invalid_AddressedTarget;
						4: 	iResponse := eTransferResponse.invalid_Index;
						5: 	iResponse := eTransferResponse.invalid_TransferValue;
						6: 	iResponse := eTransferResponse.invalid_combination;
						7:  iResponse := eTransferResponse.access_denied_DataInUse;
						8:	iResponse := eTransferResponse.no_data_empty_slot;
					END_CASE
					
				ELSE	// A different value is treated in transfer mode or the command was mirrored wrong
					// waiting for stop ack
					IF xStopPending = FALSE THEN
						iCommandNumber := 1; 			// command 'download' for the current value
						xDownloadError := FALSE;
						iResponse := eTransferResponse.transferring;
					END_IF
				END_IF
			
			ELSE // xDownloadDone = TRUE
				IF aTransferPackages[iCurrentValue].iChannel = 0 AND aTransferPackages[iCurrentValue].iAddressedTarget = 0 AND  aTransferPackages[iCurrentValue].iIndex = 0 AND  aTransferPackages[iCurrentValue].iTransferValue = 0 THEN
					// The FB is still active although all values are already downloaded
					iResponse := eTransferResponse.transfer_successful;
					xDownloadError := FALSE;
					iCommandNumber := 3; 		// do nothing (here: command 'stop', MAs remain stopped)
				ELSE
					// Another set of values was inserted to the FB without resetting the internal state with a falling edge at xExecute before
					iResponse := eTransferResponse.FB_needs_rising_edge_xExecute;
					xDownloadError := TRUE;
					iCommandNumber := 2; 		// do nothing (here: command 'exit transfer mode')
				END_IF
			END_IF
		END_IF
		
	ELSE // xInputValid = FALSE OR xInputConsistent = FALSE
		xDownloadDone := FALSE;
		xDownloadError := TRUE;
		IF iRecValveMode = 63 THEN
			iCommandNumber := 2; 				// command 'exit transfer mode'
		ELSE
			iCommandNumber := 3;				// command 'stop'
		END_IF
	END_IF
	
	xFirstCycle := FALSE;

ELSIF xExecute = FALSE AND xFirstCycle = FALSE THEN			// falling edge at input xExecute, resetting the function block
	IF iRecValveMode = 63 THEN
		iCommandNumber := 2;								// exit transfer mode
	ELSE
		xFirstCycle := TRUE;
		xDownloadDone := FALSE;
		xDownloadError := FALSE;
		xTransferComplete := FALSE;
		iCurrentValue := 0;
		xStopPending := FALSE;
		iResponse := eTransferResponse.ready_for_new_transfer;
		iCommandNumber := 0; 								// do nothing (idle)
	END_IF
		
ELSIF xExecute = FALSE AND xFirstCycle = TRUE THEN			// idle mode for the function block
	iResponse := eTransferResponse.ready_for_new_transfer;
	iCommandNumber := 0;
END_IF

CASE iCommandNumber OF
	0: // idle

	1: // download the current value, addressed and specified in the array of values
		fbWriteValueToWord(iValue := 63, iStartBit := 0, iEndBit := 5, wDataWord := awBusDataToVTEM[0]); 												// ValveMode = 63
		fbWriteValueToWord(iValue := 0, iStartBit := 6, iEndBit := 7, wDataWord := awBusDataToVTEM[0]); 												// (empty)
		fbWriteValueToWord(iValue := aTransferPackages[iCurrentValue].iChannel, iStartBit := 8, iEndBit := 12, wDataWord := awBusDataToVTEM[0]); 		// Channel
		fbWriteValueToWord(iValue := 1, iStartBit := 13, iEndBit := 15, wDataWord := awBusDataToVTEM[0]); 												// TransferControl = download
		fbWriteValueToWord(iValue := aTransferPackages[iCurrentValue].iAddressedTarget, iStartBit := 0, iEndBit := 7, wDataWord := awBusDataToVTEM[1]); 	// AddressedTarget
		fbWriteValueToWord(iValue := aTransferPackages[iCurrentValue].iIndex, iStartBit := 8, iEndBit := 15, wDataWord := awBusDataToVTEM[1]); 			// Index
		
		awBusDataToVTEM[2] := INT_TO_WORD(aTransferPackages[iCurrentValue].iTransferValue);
	
	2: // exit transfer mode
		fbWriteValueToWord(iValue := 63, iStartBit := 0, iEndBit := 5, wDataWord := awBusDataToVTEM[0]); 												// ValveMode = 63
		fbWriteValueToWord(iValue := 0, iStartBit := 6, iEndBit := 7, wDataWord := awBusDataToVTEM[0]); 												// (empty)
		fbWriteValueToWord(iValue := aTransferPackages[iCurrentValue].iChannel, iStartBit := 8, iEndBit := 12, wDataWord := awBusDataToVTEM[0]); 		// Channel
		fbWriteValueToWord(iValue := 3, iStartBit := 13, iEndBit := 15, wDataWord := awBusDataToVTEM[0]); 												// TransferControl = exit

		awBusDataToVTEM[1] := 0; 
		awBusDataToVTEM[2] := 0; 

	3: // stop all Motion Apps
		fbWriteValueToWord(iValue := 61, iStartBit := 0, iEndBit := 5, wDataWord := awBusDataToVTEM[0]); 												// ValveMode = 61
		fbWriteValueToWord(iValue := 0, iStartBit := 6, iEndBit := 15, wDataWord := awBusDataToVTEM[0]); 												// (empty)

		awBusDataToVTEM[1] := 0; 
		awBusDataToVTEM[2] := 0; 
END_CASE

END_FUNCTION_BLOCK

// Transfermode/specific_MA_config/FB_Write_config_MA_04
/// This function block can be used to download the configuration of Motion App 4 ("Model-based proportional pressure regulation").
/// The specific parameters of this Motion App are the inputs of this FB and can be defined by the user. 
/// The function block uses the transfer mode to write this configuration to the Motion Terminal
/// and indicates the state of the download process.

FUNCTION_BLOCK FB_Write_config_MA_04
VAR_INPUT
	awBusDataFromVTEM 				: ARRAY [0..2] OF WORD;		(* 6 bytes of process data received from the Motion Terminal *)
END_VAR

